(* Schneider Machine Expert - Basic project BORANG_MODUL10_LADDER_2006485775_MUHAMMAD ALFAN FUAD DZIA UL HAQ, file version 2.7.0.0 *)
(* ProjectInformations: Name=New project *)

HARDWARE
  Cpu 0: TM221CE16R
  EthernetConfiguration: NetworkName=M221, IpAllocationMode=FixedAddress, IpAddress=0.0.0.0, SubnetMask=0.0.0.0
  SerialLineConfiguration: Baud=Baud19200, Parity=ParityEven, DataBits=DataBits8, StopBits=StopBits1, PhysicalMedium=PhysicalMediumRs485, TransmissionMode=TransmissionModeModbusRtu, SlaveId=1, Addressing=SlaveAddressing
  MastTask: UsePeriodScanMode=false, PeriodScan=100
  FastTask: Period=255
  CpuBehavior: StartingMode=StartAsPreviousState, AutoSaveRamOnEeprom=true, WatchdogPeriod=250

SYMBOLS  (address, symbol, comment, settings)
  %M1         "Running"

POU New POU
  (* SectionNumber=1 *)

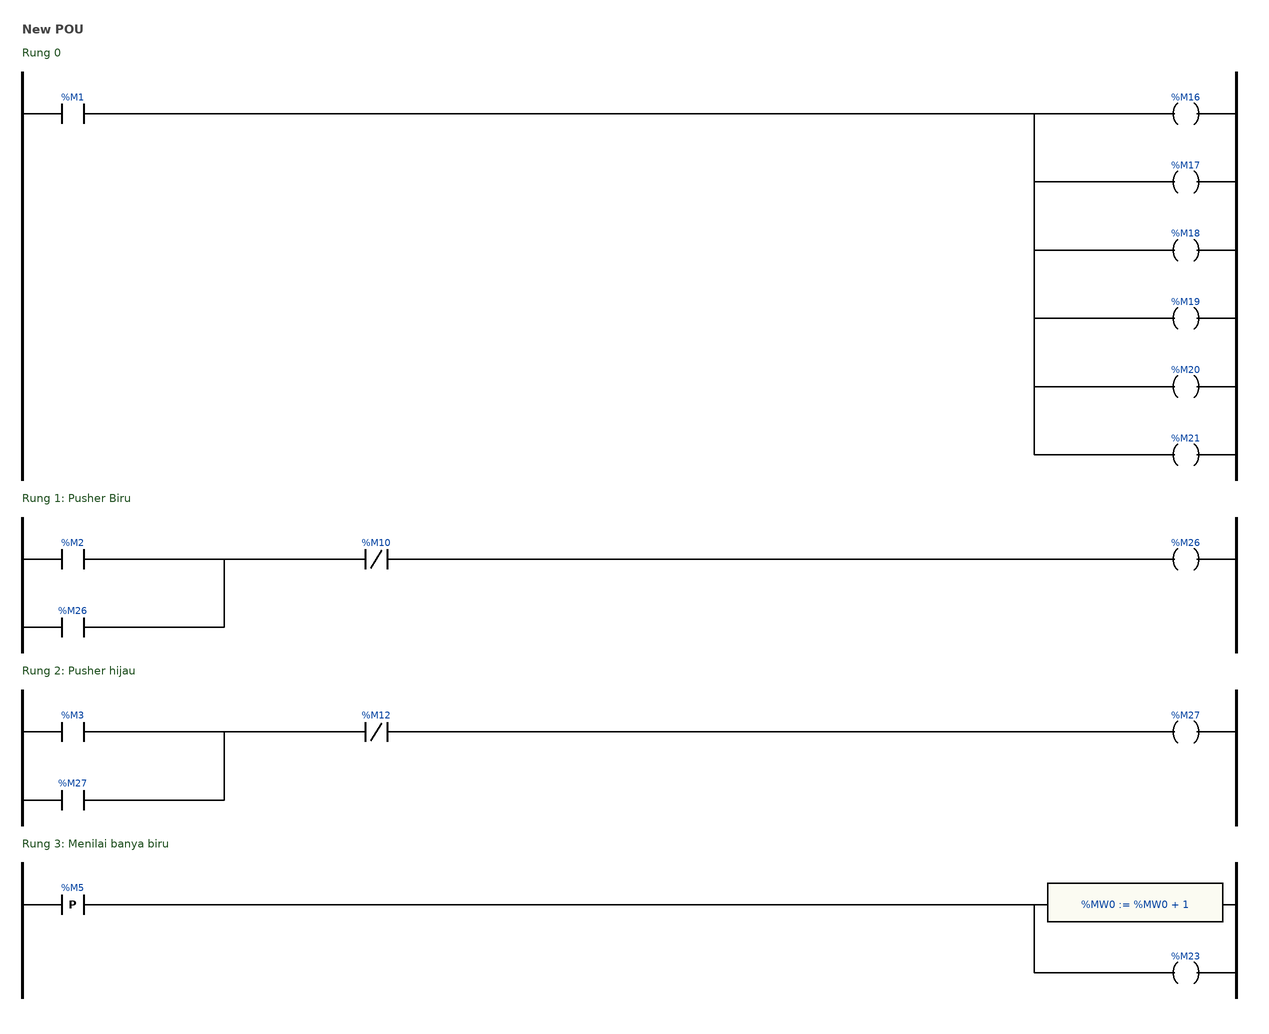

// Rung 0
  LD %M1
  ST %M16
  ST %M17
  ST %M18
  ST %M19
  ST %M20
  ST %M21
  // as ST:
  //   %M16 := %M1;
  //   %M17 := %M1;
  //   %M18 := %M1;
  //   %M19 := %M1;
  //   %M20 := %M1;
  //   %M21 := %M1;

// Rung 1: Pusher Biru
  LD %M2
  OR %M26
  ANDN %M10
  ST %M26
  // as ST:
  //   %M26 := (%M2 OR %M26) AND NOT %M10;

// Rung 2: Pusher hijau
  LD %M3
  OR %M27
  ANDN %M12
  ST %M27
  // as ST:
  //   %M27 := (%M3 OR %M27) AND NOT %M12;

// Rung 3: Menilai banya biru
  LDR %M5
  [ %MW0 := %MW0 + 1 ]
  ST %M23
  // as ST:
  //   IF RISING(%M5) THEN %MW0 := %MW0 + 1; END_IF;
  //   %M23 := RISING(%M5);
